FUNCTION_BLOCK FB_CheckString
VAR_INPUT
    data : Pers_data;
    searchString : STRING; // te zoeken string
END_VAR
VAR_OUTPUT
    found : BOOL;
END_VAR

// NOG NIET OPGELOST!!!

found := (FIND(StrToUpperA(data.Name), StrToUpperA(searchString)) <> 0) OR
         (FIND(StrToUpperA(data.Firstname), StrToUpperA(searchString)) <> 0) OR
         (FIND(StrToUpperA(data.Address), StrToUpperA(searchString)) <> 0);

END_FUNCTION_BLOCK

(* stored: Version 1.1.0.1, ProductVersion 3.1.4024.12
   POU FB_CheckString: Id {4c1954db-abef-48d3-a918-06a7c044dc84}, SpecialFunc None *)
